// TIA Portal V18 export
DATA_BLOCK "02_COM"   // DB3, F_DB
{ S7_Optimized_Access := 'TRUE'; DB_Accessible_From_OPC_UA := 'FALSE' }
VERSION : 0.1
// stored: AutoNumber true, DBAccessibleFromOPCUA false, DBAccessibleFromWebserver true
   VAR
      AlwaysFALSE : Bool;
      AlwaysTRUE : Bool;
      "No Operation" : Bool;
      "AREA 1 PB" : Bool;   // Zone cumulative: emergency push buttons - one per area that HAS E1/2 members
      "AREA 2 PB" : Bool;   // Zone cumulative: emergency push buttons - one per area that HAS E1/2 members
      "AREA 3 PB" : Bool;   // Zone cumulative: emergency push buttons - one per area that HAS E1/2 members
      "AREA 4 PB" : Bool;   // Zone cumulative: emergency push buttons - one per area that HAS E1/2 members
      "AREA 1 FDB" : Bool;   // Zone cumulative: contactor feedback - one per area with KQ members
      "AREA 2 FDB" : Bool;   // Zone cumulative: contactor feedback - one per area with KQ members
      "AREA 3 FDB" : Bool;   // Zone cumulative: contactor feedback - one per area with KQ members
      "AREA 4 FDB" : Bool;   // Zone cumulative: contactor feedback - one per area with KQ members
      "AREA 1 SAFETY_BREAKERS" : Bool;   // Zone cumulative: safety breakers - one per area with B1/2 members
      "AREA 3 SAFETY_BREAKERS" : Bool;   // Zone cumulative: safety breakers - one per area with B1/2 members
      "AREA 1 DOORS" : Bool;   // Zone cumulative: safety doors - one per area with DI1/2 members
      "AREA 3 DOORS" : Bool;   // Zone cumulative: safety doors - one per area with DI1/2 members
   END_VAR
BEGIN
END_DATA_BLOCK
